FUNCTION_BLOCK Tank_Controller (* Basic FB with empty ECC *)
  (* Standard: 61499-2 *)
  (* Version 1.0, 2025-12-25, guilh *)
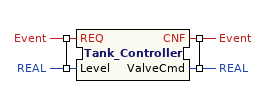
  EVENT_INPUT
    REQ WITH Level;
  END_EVENT
  EVENT_OUTPUT
    CNF WITH ValveCmd;
  END_EVENT
  VAR_INPUT
    Level : REAL;
  END_VAR
  VAR_OUTPUT
    ValveCmd : REAL;
  END_VAR
  EC_STATES
    START; (* Initial State *)
  END_STATES
END_FUNCTION_BLOCK
